(* CoDeSys 2.3.9.50 project: 3C.pr6 *)
(* Libraries: STANDARD.LB6 5.6.98 12:03:02 *)

(* POU MAIN, LD *)
PROGRAM MAIN
VAR
	SwitchA AT %IX0.0: BOOL;
	t1: TON;
	Motor AT %QX0.0: BOOL;
	SwitchB AT %IX0.1: BOOL;
	stop AT %IX0.2: BOOL;
END_VAR
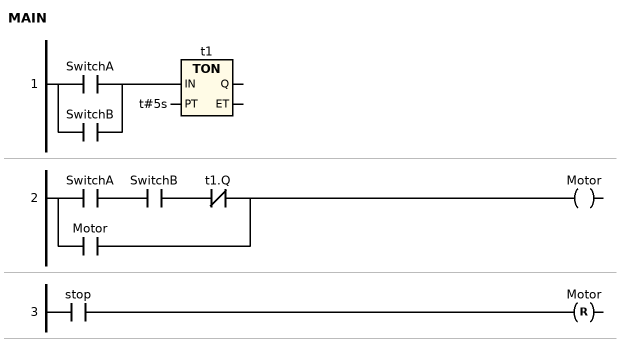
_LD_ (* Ladder Diagram *)
NETWORK 1
	{ [SwitchA] | [SwitchB] } - t1:TON(IN: *, PT: t#5s)
NETWORK 2
	{ [SwitchA] - [SwitchB] - [/t1.Q] | [Motor] } --- (Motor)
NETWORK 3
	[stop] --- (R Motor)
_END_LD_
(* the same logic as Structured Text *)
(* Network 1 *)
t1(IN := SwitchA OR SwitchB, PT := t#5s);
(* Network 2 *)
Motor := SwitchA AND SwitchB AND NOT t1.Q OR Motor;
(* Network 3 *)
IF stop THEN Motor := FALSE; END_IF;
END_PROGRAM
